// TIA Portal V18 export
TYPE "udt_Fifo"
// stored: IsFailsafeCompliant false
   STRUCT
      Entrada : Struct
         longitud : Int;
         elemento : Int;
         inserccion : Bool;
         extraccion : Bool;
         reset : Bool;
      END_STRUCT;
      Salidas : Struct
         elemento : Int;
      END_STRUCT;
      buffer : Array[0..31] of Int;
   END_STRUCT;
END_TYPE
